// TIA Portal V17 export
// export: Created 2025-08-05T09:36:00.8393853Z, ExportSetting WithDefaults, DisplayName Totally Integrated Automation Portal, DisplayVersion V17, DisplayName TIA Portal Openness, DisplayVersion V17, DisplayName TIA Portal Version Control Interface, DisplayVersion V17, DisplayName SINAMICS Startdrive Advanced, DisplayVersion V17, DisplayName SINAMICS Startdrive G130, G150, S120, S150, SINAMICS MV, S210, DisplayVersion V17, DisplayName SINAMICS Startdrive G110M, G120, G120C, G120D, G120P, G115D, DisplayVersion V17, DisplayName STEP 7 Professional, DisplayVersion V17, DisplayName STEP 7 Safety, DisplayVersion V17, DisplayName WinCC Advanced, DisplayVersion V17
TYPE "typeTeststoppSBTError"
// V 01.00
// stored: IsFailsafeCompliant false
   STRUCT
      BrakeTestParameter { S7_SetPoint := 'True'} : Bool := false;   // Störung: Bremsentest-Parameter / Fault: brake test parameter
      BrakeTestSequenceFault : Bool;   // Störung: Ablaufstörung Teststopp/Bremsentest / Fault: sequence fault test stop/brake test
      BrakeTestIntBrake : Bool;   // Störung: Bremsentest interne Bremse fehlgeschlagen / Fault: brake test internal brake failed
      BrakeTestExtBrake : Bool;   // Störung: Bremsentest externe Bremse fehlgeschlagen / Fault: brake test external brake failed
   END_STRUCT;
END_TYPE
